// TIA Portal V19 export
DATA_BLOCK "WeldReg"   // DB167
// stored: InstanceOfName WeldReg_FB, InstanceOfType FB
"WeldReg_FB"
   // VAR_INPUT
   //    AreaInterface : "AreaInterface";
   //    CIn : Struct
   //       StraightnerMaterialPresence : Bool;
   //       PinchrollMaterialPresence : Bool;
   //       PrePunchingMaterialPresence : Bool;
   //       CoilHandling_CounterValue : LReal;
   //       CoilHandling_CounterInOperation : Bool;
   //       PhaseCounterValue : LReal;
   //       PhaseCounterInOperation : Bool;
   //       WeldDone : Bool;
   //       Carriage_CounterValue : LReal;
   //       PostPunching_CounterData : "MatCountData";
   //       Manager : Struct
   //          ActTarget_P_ID : DInt;
   //          ActTarget_XStart : LReal;
   //          ActTarget_XEnd : LReal;
   //          NextTarget_P_ID : DInt;
   //          NextTarget_XStart : LReal;
   //          NextTarget_XEnd : LReal;
   //       END_STRUCT;
   //    END_STRUCT;
   // END_VAR
   // VAR_OUTPUT
   //    MachineInterface : "MachineInterface";
   //    COut : Struct
   //       WeldDoneAck : Bool;
   //       Manager : Struct
   //          ActTarget_P_ID : DInt;
   //          ActTarget_WeldPresence : Bool;
   //          ActTarget_WeldEndPos : LReal;
   //          NextTarget_P_ID : DInt;
   //          NextTarget_WeldPresence : Bool;
   //          NextTarget_WeldEndPos : LReal;
   //          WeldMIssingToFinalCut : LReal;
   //          WeldPresence : Bool;
   //       END_STRUCT;
   //    END_STRUCT;
   // END_VAR
   // VAR_IN_OUT
   //    PersistentValues : "udt_WeldReg_Pers";
   //    TO_WeldMeasInput : TO_MeasuringInput;
   // END_VAR
   // VAR
   //    Ctrl : Struct
   //       SetScrapCaseThreading : Bool;
   //       SetScrapCaseEndOfCoil : Bool;
   //       SetScrapCaseFullEmptying : Bool;
   //       WelderWriteRegExe : Bool;
   //       MeasInp_Enable : Bool;
   //    END_STRUCT;
   //    Sts : Struct
   //       InitDone : Bool;
   //       AlarmsPresence : Bool;
   //       WarningsPresence : Bool;
   //       WelderInitDone : Bool;
   //       WelderMWCounter : LReal;
   //       WelderPhaseCounter : LReal;
   //       WelderBegin_PhaseCounter : LReal;
   //       WelderEnd_PhaseCounter : LReal;
   //       WelderBegin_MWCounter : LReal;
   //       WelderEnd_MWCounter : LReal;
   //       WelderWriteRegDone : Bool;
   //       WelderEnableReg : Bool;
   //       WelderOffsetConvPhaseCounter : LReal;
   //       WelderNextScrapBegin_MWCounter : LReal;
   //       LimitOlderItem : LReal;
   //       WeldMeasInp : Struct
   //          LastID : UInt;
   //          SavedPosAxValue2 : LReal;
   //          SavedPosAxValue1 : LReal;
   //          SavedPosMatValue1 : LReal;
   //          SavedPosMatValue2 : LReal;
   //          PosBegin : LReal;
   //          PosEnd : LReal;
   //       END_STRUCT;
   //    END_STRUCT;
   //    HMI : Struct
   //       DeleteWeldRegBuffer : Bool;
   //    END_STRUCT;
   //    Alarms : Struct
   //       WeldMeasInput : "TMeasuring_Alarms";
   //    END_STRUCT;
   //    Diag : Struct
   //       WelMeasInput : "TO_Diagnostic";
   //    END_STRUCT;
   //    Warnings : Struct
   //       NoAutReady : Bool;
   //    END_STRUCT;
   //    WeldMesInp : "MeasuringInput";
   //    WeldReg_Empty : "udt_WeldReg_Item";
   //    TP_Status { S7_SetPoint := 'True'} : Int;
   // END_VAR
BEGIN
END_DATA_BLOCK
